// TIA Portal V20 export
TYPE "typeEm6Commands"
// stored: Access Published, Namespace Unit1
   STRUCT
      spare { ExternalWritable := 'False'} : Bool;
   END_STRUCT;
END_TYPE
